TYPE Kraftvariablen :
STRUCT
	Fx					:LREAL;							// Kraft in X-Richtung 
	Fy					:LREAL;							// Kraft in Y-Richtung 
	Fz					:LREAL;							// Kraft in Z-Richtung 
	Tx					:LREAL;							// Moment auf X-Achse 
	Ty					:LREAL;							// Moment auf Y-Achse 
	Tz					:LREAL;							// Moment auf Z-Achse 
END_STRUCT
END_TYPE

(* stored: Version 1.1.0.1
   DUT Kraftvariablen: Id {4040c039-1cc1-4c0a-90a7-5178cdff315a} *)
